TYPE ST_ExtAlarm :
STRUCT
	ModuleId : UDINT;
	MainErrorId : UDINT;
	SourceErrorId : UDINT;
	Message : STRING;
	Path : STRING;
	Severity : E_Severity;
	DateTime : STRING(20);	// ex: YYYYMMDDHHMMSSUU
END_STRUCT
END_TYPE

(* stored: Version 1.1.0.1, ProductVersion 3.1.4026.18
   DUT ST_ExtAlarm: Id {a176a5ca-a180-4d80-bea0-fd686a1fb7fd} *)
